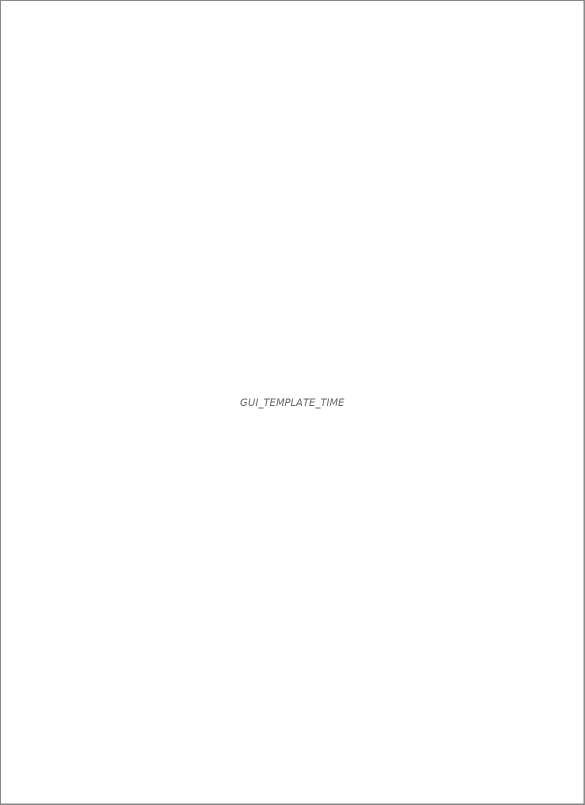
VISUALIZATION GUI_time_info  // 585x805
bVAR_IN_OUT
	
END_VAR
    Frame (0,0 585x805)
        shows GUI_TEMPLATE_TIME(m_DeviceName := 'time_info', m_Instance := MAIN.time_info)
END_VISUALIZATION

(* stored: Version 1.1.0.1, ProductVersion 3.1.4024.11
   Visu GUI_time_info: Id {9bfcbc66-9a13-457c-b41e-5c4bb95dadb7} *)
